		IF Mode = FNC_OFF 
		THEN	(* Schleifenweg Aus *)
			state 											:= 80;
		ELSE
			(* Init tmp Speicher *)
			tmpSchleifenweg 								:=
			tmpSchleifenwegPos 								:=
			tmpSchleifenwegNeg 								:= Schleifenweg;
			IF tmpSchleifenweg > 0 
			THEN
				state 										:= 20;
			ELSIF tmpSchleifenweg = 0 
			THEN
				IF Mode = FNC_NEG_DIR 
				THEN
					state 									:= 12; (* Schleifenweg nur für Neagtive Richtung ermitteln muss ermittelt werden *)
				ELSE      									
					state 									:= 10; (* Schleifenweg muss ermittelt werden *)
				END_IF
			ELSE
				ErrorID 									:= 1798;
				MemErrorState 								:= state;
				state 										:= 100;
			END_IF
		END_IF

	ELSIF NOT Execute THEN
		ReadAds	(Read := FALSE);
		WriteAds(Write := FALSE);
		Done												:= FALSE;
		Busy												:= FALSE;
		Error												:= FALSE;
		ErrorID												:= 0;
	END_IF

(* Lese Schleichweg in Pos. Richtung *)
10:
	ReadAds	(	NetId	:= '' , 
				Port	:=500, 
				IdxGrp	:=16#4000+AxID, 
				IdxOffs	:=16#301,
				LEN		:=SIZEOF(SchleichwegPos),
				DestAddr:=ADR(SchleichwegPos), 
				Read 	:= TRUE, 
				TmOut	:=T#1S );

	(* ADS Auftrag ausgeführt *)
	IF ReadAds.ERR 
	THEN
		ErrorID 											:= ReadAds.ERRID;
		MemErrorState 										:= state;
		state 												:= 100;
	ELSIF NOT ReadAds.BUSY 
	THEN
		state 												:= 11;
		ReadAds	(Read := FALSE);
	END_IF

(* Lese Bremsweg in Pos. Richtung *)
11:
	ReadAds(	NetId:= '' , 
				Port:=500, 
				IdxGrp:=16#4000+AxID, 
				IdxOffs:=16#303,
				LEN:=SIZEOF(BremswegPos),
				DestAddr:=ADR(BremswegPos), 
				Read := TRUE, 
				TmOut:=t#1s );

	(* ADS Auftrag ausgeführt *)
	IF ReadAds.ERR 
	THEN
		ErrorID 											:= ReadAds.ERRID;
		MemErrorState 										:= state;
		state 												:= 100;
	ELSIF NOT ReadAds.BUSY 
	THEN
		IF Mode = 2 
		THEN (* Schleifenweg nur für Positive Richtung ermitteln *)
			state 											:= 20;
		ELSE        										
			state 											:= 12;
		END_IF
		tmpSchleifenwegPos 									:= BremswegPos + (SchleichwegPos * 0.5);
		ReadAds	(Read := FALSE);
	END_IF

(* Lese Schleichweg in Neg. Richtung *)
12:
	ReadAds	(	NetId:= '' , 
				Port:=500, 
				IdxGrp:=16#4000+AxID, 
				IdxOffs:=16#302,
				LEN:=SIZEOF(SchleichwegNeg),
				DestAddr:=ADR(SchleichwegNeg), 
				Read := TRUE, 
				TmOut:=t#1s );

	(* ADS Auftrag ausgeführt *)
	IF ReadAds.ERR 
	THEN
		ErrorID 											:= ReadAds.ERRID;
		MemErrorState 										:= state;
		state 												:= 100;
	ELSIF NOT ReadAds.BUSY 
	THEN
		state 												:= 13;
		ReadAds	(Read := FALSE);
	END_IF

(* Lese Bremsweg in Neg. Richtung *)
13:
	ReadAds	(	NetId:= '' , 
				Port:=500, 
				IdxGrp:=16#4000+AxID, 
				IdxOffs:=16#304,
				LEN:=SIZEOF(BremswegNeg),
				DestAddr:=ADR(BremswegNeg), 
				Read := TRUE, 
				TmOut:=t#1s );

	(* ADS Auftrag ausgeführt *)
	IF ReadAds.ERR 
	THEN
		ErrorID 											:= ReadAds.ERRID;
		MemErrorState 										:= state;
		state 												:= 100;
	ELSIF NOT ReadAds.BUSY 
	THEN
		tmpSchleifenwegNeg 									:= BremswegNeg + (SchleichwegNeg * 0.5);
		ReadAds	(Read := FALSE);
		state 												:= 20;
	END_IF

(* Select Mode *)
20:
	IF Mode = FNC_OFF 
	THEN
		state 												:= 80;
	ELSIF Mode = FNC_AUTO 
	THEN (* Schleifenweg Automatik *)
		IF Istwert >= Sollwert - BremswegNeg 
		AND Istwert <= Sollwert + BremswegPos 
		THEN (* Istwert im Bremsbereich der Achse *)
			IF Istwert >= Sollwert 
			THEN (* Sollwert Positiv *)
				IF NOT (Sollwert + tmpSchleifenwegPos >= SWEndlagePos) 
				THEN (* -> Pos.Schleifenweg nicht in SoftwareEndlage Pos -> Pos. Schleifenweg *)
					tmpSchleifenweg 						:= tmpSchleifenwegPos;
					state := 30; (* Schleifenweg Ein *)
				ELSIF NOT (Sollwert - tmpSchleifenwegNeg <= SWEndlageNeg) 
				THEN
					tmpSchleifenweg 						:= tmpSchleifenwegNeg * -1 ;
					state 									:= 30; (* Schleifenweg Ein *)
				ELSE
					ErrorID 								:= 1798;
					MemErrorState 							:= state;
					state 									:= 100; (* Schleifenweg Pos,Neg liegt in SW Endlagen *)
				END_IF
			ELSIF Istwert <= Sollwert 
			THEN (* Sollwert Negativ überfahren *)
				IF NOT (Sollwert - tmpSchleifenwegNeg <= SWEndlageNeg) 
				THEN (* -> Neg.Schleifenweg nicht in SoftwareEndlage Neg -> Neg. Schleifenweg *)
					tmpSchleifenweg 						:= tmpSchleifenwegNeg * -1 ;
					state 									:= 30; (* Schleifenweg Ein *)
				ELSIF NOT (Sollwert + tmpSchleifenwegPos >= SWEndlagePos) 
				THEN
					tmpSchleifenweg := tmpSchleifenwegPos;
					state 									:= 30; (* Schleifenweg Ein *)
				ELSE
					ErrorID 								:= 1798;
					MemErrorState 							:= state;
					state 									:= 100; (* Schleifenweg Pos,Neg liegt in SW Endlagen *)
				END_IF
			ELSE
				state 										:= 80; (* Schleifenweg nicht nötig *)
			END_IF
		ELSE
			state 											:= 80; (* Schleifenweg nicht nötig *)
		END_IF
	ELSIF Mode = FNC_POS_DIR 
	THEN (* Schleifenweg Ein Positiv *)
		IF tmpSchleifenweg = 0 
		THEN
			tmpSchleifenweg 								:= tmpSchleifenwegPos;
		END_IF
		state 												:= 30; (* Schleifenweg Ein *)
	ELSIF Mode = FNC_NEG_DIR 
	THEN (* Schleifenweg Ein Neagtiv*)
		IF tmpSchleifenweg = 0 
		THEN
			tmpSchleifenweg 								:= tmpSchleifenwegNeg * -1;
		ELSE
			tmpSchleifenweg 								:= tmpSchleifenweg * -1; (* Schleifenweg Negieren *)
		END_IF
		state 												:= 30; (* Schleifenweg Ein *)
	ELSE
		ErrorID 											:= 1798;
		MemErrorState 										:= state;
		state 												:= 100;
	END_IF

(* Schleifenweg beschreiben *)
30:
	WriteAds(	NetId:= '' , 
				Port:=500, 
				IdxGrp:=16#4000+AxID, 
				IdxOffs:=16#14,
				LEN:=SIZEOF(tmpSchleifenweg),
				SrcAddr:=ADR(tmpSchleifenweg), 
				Write := TRUE, 
				TmOut:=t#1s );

	(* ADS Auftrag ausgeführt *)
	IF WriteAds.ERR 
	THEN
		ErrorID 											:= WriteAds.ERRID;
		MemErrorState 										:= state;
		state 												:= 100;
	ELSIF NOT WriteAds.BUSY 
	THEN
		WriteAds(Write := FALSE);
		state 												:= 31;
	END_IF

(* Schleifenweg Ein *)
31:
	iValue:=BOOL_TO_INT (TRUE);
	
	WriteAds(	NetId:= '' , 
				Port:=500, 
				IdxGrp:=16#4000+AxID, 
				IdxOffs:=16#13,
				LEN:=SIZEOF(iValue),
				SrcAddr:=ADR(iValue), 					
				Write := TRUE, 
				TmOut:=T#1S );

	(* ADS Auftrag ausgeführt *)
	IF WriteAds.ERR 
	THEN
		ErrorID 											:= WriteAds.ERRID;
		MemErrorState 										:= state;
		state 												:= 100;
	ELSIF NOT WriteAds.BUSY 
	THEN
		Done 												:= TRUE;
		state 												:= 0;
	END_IF

(* Schleifenweg Aus *)
80:
	iValue:=BOOL_TO_INT (FALSE);
	
	WriteAds(	NetId:= '' , 
				Port:=500, 
				IdxGrp:=16#4000+AxID, 
				IdxOffs:=16#13,
				LEN:=SIZEOF(iValue),
				SrcAddr:=ADR(iValue),
				Write := TRUE, 
				TmOut:=t#1s );

	(* ADS Auftrag ausgeführt *)
	IF WriteAds.ERR 
	THEN
		ErrorID												:= WriteAds.ERRID;
		MemErrorState 										:= state;
		state 												:= 100;
	ELSIF NOT WriteAds.BUSY 
	THEN
		Done 												:= TRUE;
		state 												:= 0;
	END_IF

(* Error State *)
100:
	Error													:= TRUE;
	state 													:= 0;
ELSE (* else case *)
	;
END_CASE

(**************************************************************************************************)

END_FUNCTION_BLOCK

// ---- POUs/PTP/03_Utilities/MMIN_TO_MMS.TcPOU
FUNCTION MMIN_TO_MMS : LREAL
VAR_INPUT
	IN														:	LREAL;
END_VAR
VAR
END_VAR

IF IN = 0.0
THEN
	MMIN_TO_MMS 											:= 0.0;
ELSE            											
	MMIN_TO_MMS 											:= IN * 1000.0 / 60.0	;
END_IF

END_FUNCTION

// ---- POUs/PTP/03_Utilities/SetOvrVelo.TcPOU
{attribute 'no_check'}
FUNCTION SetOvrVelo : LREAL
VAR_INPUT
	SetVelo													:	LREAL;
	MaxVelo													:	LREAL;
END_VAR
VAR
END_VAR

IF 	MaxVelo = 0.0 
	OR SetVelo = 0.0
THEN
	SetOvrVelo 												:= 0.0;
ELSE                										
	SetOvrVelo 												:= 100.0 / MaxVelo * SetVelo;
END_IF

END_FUNCTION

// ---- POUs/UNIT/fb_Apron/Analog_To_Slide.TcPOU
FUNCTION Analog_To_Slide : REAL
VAR_INPUT
	val	:DINT;
	dir		:INT;	//0:Btm Fold  1:Top Fold	2：Btm Fold2
END_VAR
VAR
	rel1,rel2	:REAL;
END_VAR

IF dir=1 THEN
	rel1:= LIMIT(1.0,TO_REAL(val-4992),29622);		//[0,220] [10000,30000]
	rel2:= rel1*220/(29622-4992);
ELSIF dir=2 THEN
	rel1:= LIMIT(1.0,TO_REAL(val-3150),28110);		//[0,220] [3150,30000]
	rel2:= rel1*220/(28110-3150);
ELSE
	rel1:= LIMIT(1.0,TO_REAL(val-4740),29700);		//[0,220] [10000,30000]
	rel2:= rel1*220/(29700-4740);
END_IF

Analog_To_Slide:=to_real(TRUNC((rel2) *10+0.5)/10);

END_FUNCTION

// ---- POUs/UNIT/fb_Apron/Angle_To_Analog.TcPOU
FUNCTION Angle_To_Analog : DINT
VAR_INPUT
	angle	:REAL;
		dir		:INT;	//0:Btm Fold  1:Top Fold
END_VAR
VAR
	i,j	:INT;
	rtn :DINT;
END_VAR

i:=TO_INT(angle*10)/10;
j:=TO_INT(angle*10) MOD 10;

IF dir=1 THEN
	rtn:=(AngleMap_Top[i+1]-AngleMap_Top[i])*j/10 + AngleMap_Top[i];
	;
ELSE
	rtn:=(AngleMap_Btm[i+1]-AngleMap_Btm[i])*j/10 + AngleMap_Btm[i];
	;
END_IF

Angle_To_Analog:=rtn;

END_FUNCTION

// ---- POUs/UNIT/fb_Apron/FB_SlideAbsPos.TcPOU
FUNCTION_BLOCK FB_SlideAbsPos
VAR_INPUT
	Top_Enable	:BOOL;
	Top_Para	:INT;		//Para:0  AtWorkPos ,   1,2,3     下台板滑动定位; 	Para:4   自由定位
	Top_Target	:REAL;
	Btm_Enable	:BOOL;
	Btm_Para	:INT;		//Para:0 AtWorkPos ,   1,2,3 		下台板滑动定位; 	Para:4  自由定位	
	Btm_Target	:REAL;
	Rst	:BOOL;
END_VAR
(*
Para:0  AtWorkPos ,   1,2,3,4     下台板滑动定位; Para:5   自由定位
Para:0 AtWorkPos ,    1,2,3,4 	  下台板滑动定位; Para:5  自由定位
*)
VAR_OUTPUT
	TopDone	:BOOL;
	BtmDone	:BOOL;
	bOutApronTop_SlideFWD	:BOOL;
	bOutApronTop_SlideBWD	:BOOL;
	bOutApronBtm_SlideFWD	:BOOL;
	bOutApronBtm_SlideBWD	:BOOL;
	bApronTopSlide_AtSlow , bApronBtmSlide_AtSlow: BOOL;
	
END_VAR
VAR
	tMan1,tMan2		:TON;
	iApronTopSlideAbs,iApronBtmSlideAbs: INT;
	tonTop1: Ton;
	tonBtm1: Ton;
	aa: INT;
END_VAR

IF Rst THEN
	iApronTopSlideAbs	:=50;
	iApronBtmSlideAbs	:=50;
END_IF

CASE Top_Para OF
	0:
		Top_Target	:=CNST_APRON_TOPSLIDE_POS0;
	1:
		Top_Target	:=CNST_APRON_TOPSLIDE_POS1;
	2:
		Top_Target	:=CNST_APRON_TOPSLIDE_POS2;
	3:
		Top_Target	:=CNST_APRON_TOPSLIDE_POS3;
	4,5:
		IF Top_Target>CNST_APRON_TOPSLIDE_POS3 THEN
			Top_Target	:=CNST_APRON_TOPSLIDE_POS3;
		END_IF
END_CASE
(*台板滑动定位控制*)
CASE iApronTopSlideAbs  OF
	0:
		IF Top_Enable THEN
			TopDone	:=FALSE;
			IF stFolder.Status.ApronTopFold_AtHome AND stFolder.Status.Slitter_AtHome THEN
				iApronTopSlideAbs:=1;
			ELSE
				Hmi_iArray[25]:=Hmi_iArray[25] OR 16#0001;
				iApronTopSlideAbs:=10;
			END_IF
		END_IF
	1:
		IF stFolder.ApronTop_Slide_ActPos <= Top_Target AND ABS(stFolder.ApronTop_Slide_ActPos-Top_Target)>	CNST_APRON_SLIDE_WINDOWS  THEN
			bOutApronTop_SlideFWD	:=FALSE;
			bOutApronTop_SlideBWD	:=TRUE;
			iApronTopSlideAbs	:= 10;		
		ELSIF stFolder.ApronTop_Slide_ActPos >= Top_Target AND ABS(stFolder.ApronTop_Slide_ActPos-Top_Target)>	CNST_APRON_SLIDE_WINDOWS THEN
			bOutApronTop_SlideFWD	:=TRUE;
			bOutApronTop_SlideBWD	:=FALSE;
			iApronTopSlideAbs	:= 20;		
		ELSE
			iApronTopSlideAbs	:= 50;		
		END_IF
	10:
		IF (bOutApronTop_SlideBWD AND ABS(stFolder.ApronTop_Slide_ActPos - Top_Target)<	CNST_APRON_SLIDE_WINDOWS) THEN
			IF Top_Target=0 THEN
				iApronTopSlideAbs	:= 40;					//when Target is 0, Need to Delay time ,insure arrived 0
			ELSE
				iApronTopSlideAbs	:= 50;
			END_IF
		END_IF
	20:
		IF (bOutApronTop_SlideFWD AND ABS(stFolder.ApronTop_Slide_ActPos - Top_Target)< CNST_APRON_SLIDE_WINDOWS)
			AND ((Top_Target=CNST_APRON_TOPSLIDE_POS0 AND In_sigTopApron_SlideFWD) OR Top_Target>CNST_APRON_TOPSLIDE_POS0)
			THEN
			IF Top_Target=0 THEN
				iApronTopSlideAbs	:= 40;					//when Target is 0, Need to Delay time ,insure arrived 0
			ELSE
				iApronTopSlideAbs	:= 50;
			END_IF
		END_IF
	40:
		tMan1(IN:=TRUE , PT:=T#200MS , Q=> , ET=> );			//1000
		IF tMan1.Q THEN
			iApronTopSlideAbs	:= 50;
		END_IF
	50:
		tMan1(IN:=FALSE);
		bOutApronTop_SlideFWD	:=Out_ApronTop_SlideBWD	:=FALSE;
		iApronTopSlideAbs	:=0;
		Top_Enable:=FALSE;
		TopDone	:=TRUE;
END_CASE

IF iApronTopSlideAbs>0 AND 
		((bOutApronTop_SlideFWD AND ABS(stFolder.ApronTop_Slide_ActPos-Top_Target)<CNST_APRON_TOPSLIDE_FWD_DecDis)	//30
		OR (bOutApronTop_SlideBWD AND ABS(stFolder.ApronTop_Slide_ActPos-Top_Target)<CNST_APRON_TOPSLIDE_BWD_DecDis))THEN	//35
			bApronTopSlide_AtSlow	:=TRUE;
		ELSE
			bApronTopSlide_AtSlow	:=FALSE;
		END_IF



CASE Btm_Para OF
	0:
		Btm_Target	:=CNST_APRON_BTMSLIDE_POS0;
	1:
		Btm_Target	:=CNST_APRON_BTMSLIDE_POS1;
	2:
		Btm_Target	:=CNST_APRON_BTMSLIDE_POS2;
	3:
		Btm_Target	:=CNST_APRON_BTMSLIDE_POS3;
	4,5:
		IF Btm_Target>CNST_APRON_BTMSLIDE_POS3 THEN
			Btm_Target	:=CNST_APRON_BTMSLIDE_POS3;
		END_IF
END_CASE

CASE iApronBtmSlideAbs OF
	0:		
		
		IF Btm_Enable THEN
			BtmDone	:=FALSE;
			IF stFolder.Status.ApronBtmFold_AtHome AND stFolder.Status.Slitter_AtHome  THEN
				iApronBtmSlideAbs:=1;
			ELSE
				Hmi_iArray[25]:=Hmi_iArray[25] OR 16#0004;
				iApronBtmSlideAbs:=10;
			END_IF
		END_IF
	1:
		IF stFolder.ApronBtm_Slide_ActPos <= Btm_Target AND ABS(stFolder.ApronBtm_Slide_ActPos - Btm_Target)>CNST_APRON_SLIDE_WINDOWS  THEN
			bOutApronBtm_SlideFWD	:=FALSE;
			bOutApronBtm_SlideBWD	:=TRUE;
			iApronBtmSlideAbs	:= 10;
		ELSIF stFolder.ApronBtm_Slide_ActPos >= Btm_Target AND ABS(stFolder.ApronBtm_Slide_ActPos - Btm_Target)>CNST_APRON_SLIDE_WINDOWS THEN
			bOutApronBtm_SlideFWD	:=TRUE;
			bOutApronBtm_SlideBWD	:=FALSE;
			iApronBtmSlideAbs	:= 20;
		ELSE
			iApronBtmSlideAbs	:= 50;
		END_IF
	10:
		IF (bOutApronBtm_SlideBWD AND ABS(stFolder.ApronBtm_Slide_ActPos-Btm_Target)<CNST_APRON_SLIDE_WINDOWS ) THEN
			IF Btm_Target=0 THEN
				iApronBtmSlideAbs	:= 40;					//when Target is 0, Need to Delay time ,insure arrived 0
			ELSE
				iApronBtmSlideAbs	:= 50;
			END_IF
		END_IF
	20:
		IF (bOutApronBtm_SlideFWD AND ABS(stFolder.ApronBtm_Slide_ActPos-Btm_Target)<CNST_APRON_SLIDE_WINDOWS)
			AND ((Btm_Target=CNST_APRON_BTMSLIDE_POS0 AND In_sigBtmApron_SlideFWD) OR Btm_Target>CNST_APRON_BTMSLIDE_POS0)
		 THEN
			IF Btm_Target=0 THEN
				iApronBtmSlideAbs	:= 40;					//when Target is 0, Need to Delay time ,insure arrived 0
			ELSE
				iApronBtmSlideAbs	:= 50;
			END_IF
		END_IF
	40:
		tMan2(IN:=TRUE , PT:=T#200MS , Q=> , ET=> );			//800
		IF tMan2.Q THEN
			iApronBtmSlideAbs	:= 50;
		END_IF
	50:
		tMan2(IN:=FALSE);
		bOutApronBtm_SlideFWD	:=bOutApronBtm_SlideBWD	:=FALSE;
		iApronBtmSlideAbs	:=0;
		Btm_Enable	:=FALSE;
		BtmDone	:=TRUE;
END_CASE

IF iApronBtmSlideAbs>0 AND ((bOutApronBtm_SlideFWD AND ABS(stFolder.ApronBtm_Slide_ActPos-Btm_Target)<CNST_APRON_BTMSLIDE_FWD_DecDis)		//32
	OR (bOutApronBtm_SlideBWD AND ABS(stFolder.ApronBtm_Slide_ActPos-Btm_Target)<CNST_APRON_BTMSLIDE_BWD_DecDis)) THEN	//	42
	bApronBtmSlide_AtSlow	:=TRUE;
ELSE
	bApronBtmSlide_AtSlow	:=FALSE;
END_IF
		

IF TopDone  THEN
	bOutApronTop_SlideFWD	:=bOutApronTop_SlideBWD	:=FALSE;
	stFolder.Status.ApronTopSlide_AtSlow	:=FALSE;
END_IF;
IF 	BtmDone THEN
	bOutApronBtm_SlideFWD	:=bOutApronBtm_SlideBWD	:=FALSE;
	stFolder.Status.ApronBtmSlide_AtSlow	:=FALSE;
END_IF;

tonTop1(IN:=TopDone , PT:=T#2S , Q=> , ET=> );
tonBtm1(IN:=BtmDone , PT:=T#2S , Q=> , ET=> );
IF tonTop1.Q THEN
	TopDone	:=FALSE;
END_IF;
IF tonBtm1.Q THEN 
	BtmDone	:=FALSE;
END_IF

END_FUNCTION_BLOCK

// ---- POUs/UNIT/fb_Apron/Slide_To_Analog.TcPOU
FUNCTION Slide_To_Analog : DINT
VAR_INPUT
	slide	:REAL;
	dir		:INT;	//0:Btm Fold  1:Top Fold
	
END_VAR
VAR
	i,j	:INT;
	rtn :DINT;
END_VAR

i:=TO_INT(slide*10)/10;
j:=TO_INT(slide*10) MOD 10;

IF dir=1 THEN					
	rtn:= TO_INT(slide*(29622-4992)/220+4992);			//[0,220] [4992,29622]
ELSE
	rtn:= TO_INT(slide*(29700-4740)/220+4740);			//[0,220] [4740,29700]
END_IF

Slide_To_Analog:=rtn;

END_FUNCTION

// ---- POUs/UNIT/fb_BackGauge/FB_BGAbsPos.TcPOU
FUNCTION_BLOCK FB_BGAbsPos
VAR_INPUT
	Ex			:BOOL;
	Mode		:INT;	(*1:直接定位	2:后退式定位*)
	TargetPos	:LREAL;
	ActPos 		:LREAL;
	GripType	:INT;	(*0:PUSH 1:Grip  2:OverGrip 3:Observe  4:Home*)
	GripOPEN	:BOOL;	(*false:保持原状态  true：打开后定位*)
	Velo		:LREAL;
	Rst			:BOOL;
	RstDone	:BOOL;
END_VAR
VAR_OUTPUT
	Busy	:BOOL;
	Done	:BOOL;
END_VAR
VAR_IN_OUT
	Ax			:Axis_PTPV3_CoE;
END_VAR
VAR
	iPTP: INT;
	GripAttach	:REAL;
	ton1: Ton;
	ton2: Ton;
	rTemp0: REAL;
END_VAR

IF Rst THEN
	iPTP	:=121;
END_IF

CASE iPTP OF
	0:
		IF Ex THEN
			iPTP	:=1;
			Done	:=FALSE;
		END_IF
	1:
		Ax.NoAction();
		IF GripOPEN THEN
			stFolderCom.paraBackGauge_Grip :=1;
		END_IF
		IF mode=1 THEN
			iPTP	:=100;
		ELSIF mode=2 THEN
			iPTP	:=10;
		END_IF;
	10:
		Out_GripperDatum_S0	:=Out_GripperDatum_S1	:=TRUE;
		ton2(IN:=TRUE , PT:=T#1S , Q=> , ET=> );
		IF ton2.Q THEN
			iPTP:=11;
			ton2(IN:=FALSE);
		END_IF;
	11:
		Out_GripperDatum_S0	:=Out_GripperDatum_S1	:=TRUE;
		//rTemp0	:=stFolderPara.BackGaugeMaxPos-stFolder.BackGauge_M_ActPos;		//此处需要修改
		rTemp0	:=stFolderPara.BackGaugeMaxPos-MAIN.fbMachine._ActBG_Target;
		iPTP:=12;
	12:
		Out_GripperDatum_S0	:=Out_GripperDatum_S1	:=TRUE;
		Ax.Motion.Velo:=Velo;
		Ax.Motion.Target:= LIMIT(0, rTemp0 - 100.0,1210);
		Ax.Motion.MoveAbs(TRUE);
		IF  Ax.Motion.Done OR ABS(Ax.Motion.Target-Ax.ref.NcToPlc.ActPos)<0.1 THEN
			iPTP:=13;
		END_IF
	13:
		Ax.NoAction();
		iPTP:=20;
	20:
		IF GripType =1 THEN
			stFolderCom.paraBackGauge_GripType := 1;
		ELSIF GripType =2 THEN
			stFolderCom.paraBackGauge_GripType := 2;
		ELSIF GripType =4 THEN
			stFolderCom.paraBackGauge_GripType := 4;
		END_IF
		iPTP:=100;
	100:
		IF GripType =1 THEN
			GripAttach	:=CNST_BACKGAUGE_ATTACH_GRIP;
		ELSIF GripType =2 THEN
			GripAttach	:=CNST_BACKGAUGE_ATTACH_OVERGRIP;
		ELSIF GripType =4 THEN
			GripAttach	:=CNST_BACKGAUGE_ATTACH_BACK;
		ELSE
			GripAttach	:=0;
			stFolderCom.paraBackGauge_Grip := 0;
		END_IF
		Ax.Motion.MoveAbs(FALSE);
		iPTP:=101;
	101:
		IF TargetPos> ActPos THEN
			iPTP:=110;
		ELSE
			iPTP:=120;
		END_IF
	110:
		Ax.Motion.Velo:=Velo;
		IF stFolder.SlitterRef THEN
			Ax.Motion.Target:= LIMIT(-20, stFolderPara.BackGaugeMaxPos - TargetPos + stFolderPara.SlitterOffset + GripAttach -20,1210);
		ELSE
			Ax.Motion.Target:= LIMIT(-20, stFolderPara.BackGaugeMaxPos - TargetPos + GripAttach - 20,1210);
		END_IF;
		Ax.Motion.MoveAbs(TRUE);
		IF  Ax.Motion.Done OR ABS(Ax.Motion.Target-Ax.ref.NcToPlc.ActPos)<0.1  THEN
			iPTP:=111;
		END_IF
	111:
		Ax.NoAction();
		iPTP:=120;
	120:
		Ax.Motion.Velo:=Velo;
		IF stFolder.SlitterRef THEN		(*以分条还是折弯位为基准*)
			Ax.Motion.Target:= LIMIT(-20, stFolderPara.BackGaugeMaxPos - TargetPos + stFolderPara.SlitterOffset + GripAttach,1210);
		ELSE
			Ax.Motion.Target:= LIMIT(-20, stFolderPara.BackGaugeMaxPos - TargetPos + GripAttach,1210);
		END_IF
		
		Ax.Motion.MoveAbs(TRUE);
		//Ax.Motion.Halt(TRUE);
		
		IF  Ax.Motion.Done OR abs(Ax.Motion.Target-Ax.ref.NcToPlc.ActPos)<0.1 THEN
			iPTP:=121;			
		END_IF
	121:
		Ax.NoAction();
		iPTP:=0;
		Done:=TRUE;
		Ex:=FALSE;
END_CASE

Busy	:=iPTP>0;
IF RstDone THEN
	Done:=FALSE;
END_IF
(*
ton1(IN:=Done , PT:=T#1S , Q=> , ET=> );
IF ton1.Q THEN 
	Done:=FALSE;
	
END_IF
*)

END_FUNCTION_BLOCK

// ---- POUs/UNIT/fb_Clamp/Anolog_To_Height.TcPOU
FUNCTION Anolog_To_Height : real
VAR_INPUT
	value	:DINT;
END_VAR
VAR
	i	:INT;
	rel1,rel2	:REAL;
END_VAR

i:=0;

WHILE (HeightMap[i]<value AND HeightMap[i]>0) DO
	i:=i+1;
END_WHILE
i	:=LIMIT(1,i,380);
rel1:= TO_REAL(value-HeightMap[i-1]);
rel2:= rel1/LIMIT(1.0,TO_REAL(HeightMap[i]-HeightMap[i-1]),10000);

Anolog_To_Height:=LIMIT(0,TO_REAL(i-1)+rel2,380);

END_FUNCTION

// ---- POUs/UNIT/fb_Clamp/FB_ClampJog.TcPOU
FUNCTION_BLOCK FB_ClampJog
VAR_INPUT
	Rst	:BOOL;
END_VAR
VAR_OUTPUT
END_VAR
VAR
	iClampDn1,iClampUp1	:INT;
	rtClampDn	:R_TRIG;
	rtClampUp	:R_TRIG;
	flag00,flag01: BOOL;
	tonPedalClampDn	:TON;
	tonPedalClampUp	:TON;
	flag02: BOOL;
	bUnClamp: BOOL;
	bClamp: BOOL;
END_VAR

IF Rst THEN
	iClampDn1	:=30;	iClampUp1	:=2;
END_IF

flag00:=stFolder.Status.Slitter_AtHome AND stFolder.Status.ApronTopFold_AtHome AND stFolder.Status.ApronBtmFold_AtHome;
bUnClamp:= pedal_UnClamp;
bClamp	:= pedal_Clamp;

flag01:=flag00 AND stFolder.Status.Table_AtHome;
tonPedalClampDn(IN:=bClamp AND NOT bUnClamp , PT:=T#500MS , Q=> , ET=> );
tonPedalClampUp(IN:=NOT bClamp AND bUnClamp , PT:=T#500MS , Q=> , ET=> );
rtClampDn(CLK:=tonPedalClampDn.Q , Q=> );
rtClampUp(CLK:=tonPedalClampUp.Q , Q=> );


//flag00:=TRUE;
//flag01:=TRUE;
CASE iClampDn1 OF
	0:
		IF rtClampDn.Q AND flag01 THEN
			IF NOT stFolder.Status.Clamp_LtHalfPoint THEN
				iClampDn1	:=10;
			ELSIF stFolder.Status.Clamp_LtHalfPoint THEN
				iClampDn1	:=20;
			ELSE
				iClampDn1	:=30;
			END_IF
		END_IF
	10:
		Out_ClampDown	:=TRUE;
		Out_ClampUp		:=FALSE;
		iClampDn1	:=SEL(NOT bClamp OR stFolder.Status.Clamp_LtHalfPoint,10,30);
	20:
		Out_ClampDown	:=TRUE;
		Out_ClampUp		:=FALSE;
		//flag01	:= (stFolder.Status.Clamp_AtZeroPoint AND stFolder.Status.Clamp_AtPressPoint);
		//flag01	:= (stFolder.Status.Clamp_AtZeroPoint);
		iClampDn1	:=SEL((NOT bClamp OR flag02),20,30);
	30:
		Out_ClampDown:= Out_ClampUp :=FALSE;
		iClampDn1	:=0;
END_CASE

CASE iClampUp1 OF
	0: 
		IF flag00 AND rtClampUp.Q THEN
			iClampUp1	:=1;
			iClampDn1	:=0;
		END_IF
		
	1:
		Out_ClampUp		:=TRUE;
		Out_ClampDown	:=FALSE;
		iClampUp1	:=SEL(NOT bUnClamp OR stFolder.ClampHt_ActPos>=stFolderPara.Clamp_MaxPos,1,2);
//		iClampUp1	:=SEL(NOT bUnClamp ,1,2);
	2:
		Out_ClampUp	:= Out_ClampDown	:=FALSE;
		iClampUp1	:=0;
		
		
END_CASE

END_FUNCTION_BLOCK

// ---- POUs/UNIT/fb_Clamp/FB_ClampLock.TcPOU
FUNCTION_BLOCK FB_ClampLock
VAR_INPUT
	Ex		:BOOL;
	para	:INT;	(* 0:Clamp_LowPos  1:Clamp_MidPos  2:Clamp_HighPos	3:Clamp_MaxPos	4:ClampHalfPos	5:Close*)					
	Rst	:BOOL;
END_VAR
VAR_OUTPUT
	Done	:BOOL;
END_VAR
VAR
	tmpTarget: REAL;
	iClampDn2: INT;
	tonDone: TON;
	ton1: Ton;
END_VAR

IF Rst THEN
	iClampDn2	:=5;
END_IF

CASE para OF
	0:
		tmpTarget	:=stFolderPara.Clamp_LowPos;
	1:
		tmpTarget	:=stFolderPara.Clamp_MidPos;
	2:
		tmpTarget	:=stFolderPara.Clamp_HighPos;
	3:
		tmpTarget	:=stFolderPara.Clamp_MaxPos;
	4:
		tmpTarget	:=stFolderPara.ClampHalfPos;
	5:
		tmpTarget	:=CONST_CLAMP_POS_CALIBRATION;
	6:
		tmpTarget	:=0;
	10..200:
		tmpTarget	:=para;
END_CASE


CASE iClampDn2 OF
	0:
		IF Ex THEN
			iClampDn2	:=1;
				ton1(IN:=FALSE);
			Done	:=FALSE;
		ELSE
			Done	:=FALSE;
		END_IF;
	1:
		Out_ClampUp		:=FALSE;
		Out_ClampDown	:= TRUE;
		
		IF (para<6 AND stFolder.ClampHt_ActPos<=tmpTarget)
			OR (para=6  AND stFolder.Status.Clamp_AtZeroPoint AND stFolder.Status.Clamp_AtPressPoint)
 			OR (para<>6 and stFolder.ClampHt_ActPos<=tmpTarget)
			OR pedal_UnClamp THEN
				iClampDn2	:=2;
		END_IF
	2:
		Out_ClampDown:= FALSE;
		Out_ClampUp := pedal_UnClamp;
		ton1(IN:= NOT Out_ClampDown AND NOT Out_ClampUp , PT:=T#100MS , Q=> , ET=> );
		IF	ton1.Q THEN
			iClampDn2	:=3;
		END_IF;
	3:
		iClampDn2	:=4;
	4:
		iClampDn2	:=5;
	5:
		
		ton1(IN:=FALSE);
		Done	:=TRUE;
		Ex:=FALSE;
END_CASE

tonDone(IN:=Done , PT:=T#200MS , Q=> , ET=> );

IF tonDone.Q THEN
	Done	:=FALSE;
	iClampDn2	:=0;
	ton1(IN:=FALSE);Ex:=FALSE;
END_IF

END_FUNCTION_BLOCK

// ---- POUs/UNIT/fb_Slitter/FB_SlitterAct.TcPOU
FUNCTION_BLOCK FB_SlitterAct
VAR_INPUT
	ExHome	:BOOL;
END_VAR
VAR_OUTPUT
	Done	:BOOL;
END_VAR
VAR
	iManSlitStep	:INT;
	tonPedalSlite,tonPedalSliteBack	:TON;
	bTmp1: BOOL;
	bManSlitRunning: BOOL;
	i: INT;
	tonDone	:TON;
	bSlitterFwd: BOOL;
	bSlitterBwd: BOOL;
	bOutSlitterFwd: BOOL;
	bOutSlitterBwd: BOOL;
	rtPedalSlit,rtPedalSlitBack		:R_TRIG;
	rtTonPedalSlit,rtTonPedalSlitBack	:R_TRIG;
	iManStop: INT;
	tonStop1: TON;
	bSlitter: BOOL;
	bSlitterBack: BOOL;
END_VAR

bSlitter:=pedal_Slitter;
bSlitterBack:=pedal_SlitterBack;

rtPedalSlit(CLK:=bSlitter AND NOT In_sigSlitLmt1 AND NOT bOutSlitterBwd  , Q=> );
rtPedalSlitBack(CLK:=NOT bSlitter AND bSlitterBack AND NOT In_sigSlitLmt0  , Q=> );
tonPedalSlite(IN:=bSlitter AND NOT bSlitterBack , PT:=T#600MS , Q=> , ET=> );
tonPedalSliteBack(IN:=NOT bSlitter AND bSlitterBack , PT:=T#600MS , Q=> , ET=> );
rtTonPedalSlit(CLK:=tonPedalSlite.Q , Q=> );
rtTonPedalSlitBack(CLK:=tonPedalSliteBack.Q, Q=> );

IF (rtPedalSlit.Q OR rtPedalSlitBack.Q OR b_sigLC_VShort) AND bManSlitRunning THEN
	iManStop:=1;
ELSIF rtTonPedalSlit.Q  THEN
	bManSlitRunning	:=TRUE;
	iManSlitStep	:=0;
ELSIF rtTonPedalSlitBack.Q  OR Hmi_bArray[44] OR ExHome THEN
	bManSlitRunning	:=TRUE;
	iManSlitStep	:=100;
END_IF



CASE iManSlitStep OF
	0:
		//bTmp1 :=(In_sigBtmApron_SlideFWD AND In_sigBtmApron_FoldHome AND In_sigTopApron_FoldHome AND NOT In_sigTopApron_SlideFWD) ;
		bTmp1 :=stFolder.Status.ApronBtmSlide_AtWork AND stFolder.Status.ApronBtmFold_AtHome AND stFolder.Status.ApronTopFold_AtHome AND NOT stFolder.Status.ApronTopSlide_AtWork AND stFolder.Status.Clamp_AtZeroPoint;
		IF (rtTonPedalSlit.Q OR Hmi_bArray[83]) AND bTmp1 THEN		//Hmi_bArray[83] Slitter to Orgin
			IF stFolder.Status.SlitterAtSlow THEN
				iManSlitStep	:=11;
			ELSE
				iManSlitStep	:=2;
			END_IF
		END_IF
	2:
		bManSlitRunning	:=TRUE;
		iManSlitStep	:=10;
	10:
		bOutSlitterFwd	:=bManSlitRunning;
		bOutSlitterBwd	:=FALSE;
		iManSlitStep	:=SEL(In_sigSlitSlw1 OR In_sigSlitLmt1 ,10,11);
	11:
		bOutSlitterFwd	:=bManSlitRunning;
		bOutSlitterBwd	:=FALSE;
		stFolder.Status.SlitterAtSlow	:=TRUE;
		iManSlitStep	:=SEL(In_sigSlitLmt1  ,11,12);
	12:
		stFolder.Status.SlitterAtSlow	:=FALSE;
		iManSlitStep	:=100;
	100:	(*back home返回*)
		IF stFolder.Status.SlitterAtSlow THEN
				iManSlitStep	:=102;
			ELSE
				iManSlitStep	:=101;
		END_IF
	101:
		bOutSlitterFwd	:=FALSE;
		bOutSlitterBwd	:=bManSlitRunning;
		iManSlitStep	:=SEL(In_sigSlitSlw0 OR In_sigSlitLmt0 ,101,102);
	102:
		bOutSlitterFwd	:=FALSE;
		bOutSlitterBwd	:=bManSlitRunning;
		stFolder.Status.SlitterAtSlow	:=TRUE;
		iManSlitStep	:=SEL(In_sigSlitLmt0 ,102,110);
	110:
		bOutSlitterFwd	:=bOutSlitterBwd	:= FALSE;
		stFolder.Status.SlitterAtSlow	:=FALSE;
		Done	:=TRUE;
		iManSlitStep	:=0;
		bManSlitRunning	:=FALSE;
END_CASE

tonDone(IN:=Done , PT:=T#1S , Q=> , ET=> );
IF tonDone.Q THEN 
	Done	:=FALSE;
END_IF

//********** suddenly stopping during cutting ,low speed process  *****************/
tonStop1(IN:=iManStop=1 , PT:=T#200MS , Q=> , ET=> );
CASE iManStop OF
	0:;
	1:
		stFolder.Status.SlitterAtSlow	:=TRUE;
		iManStop	:=SEL(tonStop1.Q ,1,2);
	2:
		stFolder.Status.SlitterAtSlow	:=FALSE;
		bManSlitRunning	:=FALSE;
		iManStop	:=0;
END_CASE

END_FUNCTION_BLOCK

// ---- GlobalTextList.TcGTLO
TEXTLIST GlobalTextList
  661 = '\n%s'
  55 = ' command Products: %i'
  49 = '%s'
  679 = '%s\n'
  54 = 'A C C I D E N T'
  18 = 'Abort'
  33 = 'Aborted'
  34 = 'Aborting'
  526 = 'Auto'
  779 = 'AutoSlitter'
  61 = 'Average MachSpeed: %5.2f Package/min'
  16 = 'Clear'
  32 = 'Clearing'
  17 = 'Command'
  38 = 'Complete'
  39 = 'Completing'
  58 = 'CurrentMachSpeed:%5.2f Package/min'
  50 = 'Detection\nof metal'
  68 = 'Do you want to change tp production mode?'
  23 = 'Execute'
  19 = 'Execute\nComplete'
  59 = 'Finished Metalboxes: %i'
  60 = 'Finished Plasticboxes: %i'
  56 = 'Finished Products: %i '
  25 = 'Held'
  12 = 'Hold'
  26 = 'Holding'
  21 = 'Idle'
  4 = 'Invalid'
  51 = 'Light\nsensor'
  6 = 'Mantainance'
  7 = 'Manual'
  52 = 'Move belt\n+'
  53 = 'Move to\nwork position'
  3 = 'No'
  5 = 'Production'
  9 = 'Reset'
  57 = 'Reset the Visu'
  30 = 'Reseting'
  36 = 'SC'
  492 = 'SemiAuto'
  62 = 'Seperated Boxes: %i'
  906 = 'simiAuto'
  10 = 'Start'
  22 = 'Starting'
  67 = 'State Model\n%s'
  11 = 'Stop'
  31 = 'Stopped'
  35 = 'Stopping'
  14 = 'Suspend'
  28 = 'Suspended'
  29 = 'Suspending'
  13 = 'Unhold'
  24 = 'Unholding'
  20 = 'Unit Mode'
  37 = 'Unsuspend'
  27 = 'Unsuspending'
  15 = 'Unuspend'
  8 = 'UserMode 1'
  1 = 'Yes'
  2 = 'Yes, with Reset'
END_TEXTLIST

// ---- VISUs/VISUs/Templates/VIS_TemplatePMLStateModel.TcVIS
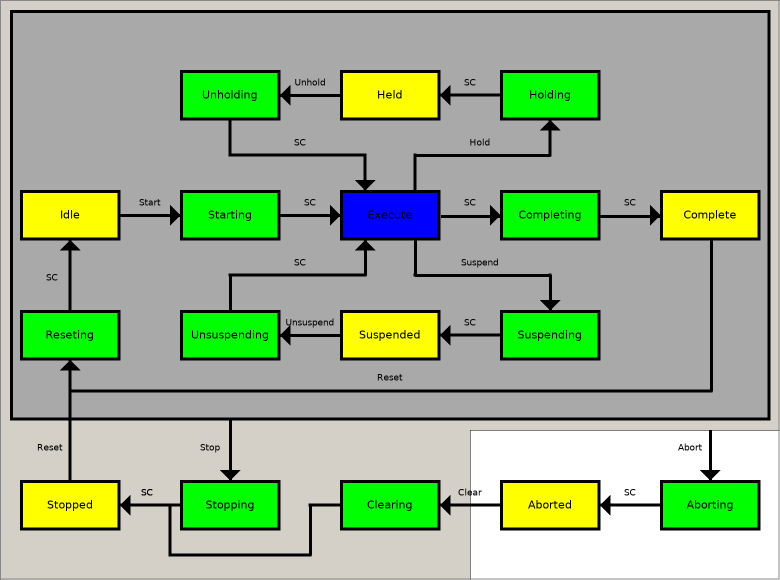
VISUALIZATION VIS_TemplatePMLStateModel  // 780x580
VAR_INPUT
	ePMLUnitMode		: DINT;
	ePMLState			: DINT;
END_VAR
    Polygon (0,0) (780,0) (780,430) (470,430) (470,580) (0,580)
    Rectangle (10,10 760x410)
    Polyline (415,190) (415,155) (550,155) (550,95) (440,95), invisible if: stPMLUnitModeConfiguration[ePMLUnitMode].aStateDisabled[11]
    Polyline (365,190) (365,155) (230,155) (230,95) (340,95), invisible if: stPMLUnitModeConfiguration[ePMLUnitMode].aStateDisabled[11]
    Polyline (415,240) (415,275) (550,275) (550,335) (440,335), invisible if: stPMLUnitModeConfiguration[ePMLUnitMode].aStateDisabled[5]
    Polyline (365,240) (365,275) (230,275) (230,335) (340,335), invisible if: stPMLUnitModeConfiguration[ePMLUnitMode].aStateDisabled[5]
    Polyline (710,430) (710,505) (310,505) (310,555) (170,555) (170,505) (70,505) (70,215) (340,215)
    RoundedRectangle (20,190 100x50), "Idle", colour toggle: (ePMLState = 4), invisible if: stPMLUnitModeConfiguration[ePMLUnitMode].aStateDisabled[4]
    RoundedRectangle (180,190 100x50), "Starting", colour toggle: (ePMLState = 3), invisible if: stPMLUnitModeConfiguration[ePMLUnitMode].aStateDisabled[3]
    RoundedRectangle (340,190 100x50), "Execute", colour toggle: (ePMLState = 6)
    RoundedRectangle (180,70 100x50), "Unholding", colour toggle: (ePMLState = 12), invisible if: stPMLUnitModeConfiguration[ePMLUnitMode].aStateDisabled[12]
    RoundedRectangle (340,70 100x50), "Held", colour toggle: (ePMLState = 11), invisible if: stPMLUnitModeConfiguration[ePMLUnitMode].aStateDisabled[11]
    RoundedRectangle (500,70 100x50), "Holding", colour toggle: (ePMLState = 10), invisible if: stPMLUnitModeConfiguration[ePMLUnitMode].aStateDisabled[10]
    RoundedRectangle (180,310 100x50), "Unsuspending", colour toggle: (ePMLState = 14), invisible if: stPMLUnitModeConfiguration[ePMLUnitMode].aStateDisabled[14]
    RoundedRectangle (340,310 100x50), "Suspended", colour toggle: (ePMLState = 5), invisible if: stPMLUnitModeConfiguration[ePMLUnitMode].aStateDisabled[5]
    RoundedRectangle (500,310 100x50), "Suspending", colour toggle: (ePMLState = 13), invisible if: stPMLUnitModeConfiguration[ePMLUnitMode].aStateDisabled[13]
    RoundedRectangle (20,310 100x50), "Reseting", colour toggle: (ePMLState = 15), invisible if: stPMLUnitModeConfiguration[ePMLUnitMode].aStateDisabled[15]
    RoundedRectangle (20,480 100x50), "Stopped", colour toggle: (ePMLState = 2)
    RoundedRectangle (340,480 100x50), "Clearing", colour toggle: (ePMLState = 1), invisible if: stPMLUnitModeConfiguration[ePMLUnitMode].aStateDisabled[1]
    RoundedRectangle (500,480 100x50), "Aborted", colour toggle: (ePMLState = 9)
    RoundedRectangle (660,480 100x50), "Aborting", colour toggle: (ePMLState = 8), invisible if: stPMLUnitModeConfiguration[ePMLUnitMode].aStateDisabled[8]
    Polygon (550,120) (540,130) (560,130), invisible if: stPMLUnitModeConfiguration[ePMLUnitMode].aStateDisabled[10]
    Polygon (365,240) (355,250) (375,250), invisible if: stPMLUnitModeConfiguration[ePMLUnitMode].aStateDisabled[5]
    Polygon (70,240) (60,250) (80,250), invisible if: stPMLUnitModeConfiguration[ePMLUnitMode].aStateDisabled[4]
    Polygon (70,360) (60,370) (80,370), invisible if: stPMLUnitModeConfiguration[ePMLUnitMode].aStateDisabled[15]
    Polygon (440,95) (450,105) (450,85), invisible if: stPMLUnitModeConfiguration[ePMLUnitMode].aStateDisabled[11]
    Polygon (280,95) (290,105) (290,85), invisible if: stPMLUnitModeConfiguration[ePMLUnitMode].aStateDisabled[12]
    Polygon (440,335) (450,345) (450,325), invisible if: stPMLUnitModeConfiguration[ePMLUnitMode].aStateDisabled[5]
    Polygon (280,335) (290,345) (290,325), invisible if: stPMLUnitModeConfiguration[ePMLUnitMode].aStateDisabled[14]
    Polygon (600,505) (610,515) (610,495)
    Polygon (440,505) (450,515) (450,495), invisible if: stPMLUnitModeConfiguration[ePMLUnitMode].aStateDisabled[1]
    Polygon (120,505) (130,515) (130,495)
    Polygon (180,215) (170,225) (170,205), invisible if: stPMLUnitModeConfiguration[ePMLUnitMode].aStateDisabled[3]
    Polygon (340,215) (330,225) (330,205)
    Polygon (500,215) (490,225) (490,205), invisible if: stPMLUnitModeConfiguration[ePMLUnitMode].aStateDisabled[16]
    Polygon (660,215) (650,225) (650,205), invisible if: stPMLUnitModeConfiguration[ePMLUnitMode].aStateDisabled[17]
    Polygon (375,180) (365,190) (355,180), invisible if: stPMLUnitModeConfiguration[ePMLUnitMode].aStateDisabled[11]
    Polygon (560,300) (550,310) (540,300), invisible if: stPMLUnitModeConfiguration[ePMLUnitMode].aStateDisabled[13]
    Polygon (720,470) (710,480) (700,470), invisible if: stPMLUnitModeConfiguration[ePMLUnitMode].aStateDisabled[8]
    Polygon (240,470) (230,480) (220,470), invisible if: stPMLUnitModeConfiguration[ePMLUnitMode].aStateDisabled[7]
    Polyline (230,420) (230,505) (150,505)
    RoundedRectangle (180,480 100x50), "Stopping", colour toggle: (ePMLState = 7), invisible if: stPMLUnitModeConfiguration[ePMLUnitMode].aStateDisabled[7]
    Label (440,135 80x15), "Hold", invisible if: stPMLUnitModeConfiguration[ePMLUnitMode].aStateDisabled[11]
    Label (260,135 80x15), "SC", invisible if: stPMLUnitModeConfiguration[ePMLUnitMode].aStateDisabled[12]
    Label (430,75 80x15), "SC", invisible if: stPMLUnitModeConfiguration[ePMLUnitMode].aStateDisabled[10]
    Label (270,75 80x15), "Unhold", invisible if: stPMLUnitModeConfiguration[ePMLUnitMode].aStateDisabled[11]
    Label (270,315 80x15), "Unsuspend", invisible if: stPMLUnitModeConfiguration[ePMLUnitMode].aStateDisabled[5]
    Label (430,315 80x15), "SC", invisible if: stPMLUnitModeConfiguration[ePMLUnitMode].aStateDisabled[13]
    Label (440,255 80x15), "Suspend", invisible if: stPMLUnitModeConfiguration[ePMLUnitMode].aStateDisabled[5]
    Label (260,255 80x15), "SC", invisible if: stPMLUnitModeConfiguration[ePMLUnitMode].aStateDisabled[14]
    Label (270,195 80x15), "SC", invisible if: stPMLUnitModeConfiguration[ePMLUnitMode].aStateDisabled[3]
    Label (590,195 80x15), "SC", invisible if: stPMLUnitModeConfiguration[ePMLUnitMode].aStateDisabled[16]
    Label (430,195 80x15), "SC", invisible if: stPMLUnitModeConfiguration[ePMLUnitMode].aStateDisabled[17]
    Label (430,485 80x15), "Clear"
    Label (590,485 80x15), "SC", invisible if: stPMLUnitModeConfiguration[ePMLUnitMode].aStateDisabled[8]
    Label (107,485 80x15), "SC", invisible if: stPMLUnitModeConfiguration[ePMLUnitMode].aStateDisabled[1]
    Label (350,370 80x15), "Reset", invisible if: stPMLUnitModeConfiguration[ePMLUnitMode].aStateDisabled[17]
    Label (10,440 80x15), "Reset", invisible if: stPMLUnitModeConfiguration[ePMLUnitMode].aStateDisabled[4]
    Label (170,440 80x15), "Stop"
    Label (650,440 80x15), "Abort"
    Label (12,270 80x15), "SC", invisible if: stPMLUnitModeConfiguration[ePMLUnitMode].aStateDisabled[15]
    Label (110,195 80x15), "Start"
    Label (107,485 80x15), "SC", invisible if: stPMLUnitModeConfiguration[ePMLUnitMode].aStateDisabled[7]
    Polyline (441,216) (711,216) (711,391) (71,391), invisible if: stPMLUnitModeConfiguration[ePMLUnitMode].aStateDisabled[17]
    RoundedRectangle (660,190 100x50), "Complete", colour toggle: (ePMLState = 17), invisible if: stPMLUnitModeConfiguration[ePMLUnitMode].aStateDisabled[17]
    RoundedRectangle (500,190 100x50), "Completing", colour toggle: (ePMLState = 16), invisible if: stPMLUnitModeConfiguration[ePMLUnitMode].aStateDisabled[16]
END_VISUALIZATION
